PROGRAM LOADINGLOGIC
VAR
END_VAR


(*LOGIC TO DEFINE WHETHER THE MOBILE ATTACHMENT IS LOWERED PROPERLY IN THE GROUND*)
IF MOBILEHOIST.FLOORPOSITION_SWITCH1 AND MOBILEHOIST.FLOORPOSITION_SWITCH2 THEN
	
	MOBILEHOIST.LOWERED_PROPERLY 			:= TRUE;
	MOBILEHOIST.LOWERED_IMPROPERLY			:= FALSE;
	MOBILEHOIST.RAISED_PROPERLY				:= FALSE;
	
(*LOGIC TO DEFINE WHETHER THE MOBILE ATTACHMENT IS IMPROPERLY LOWERED*)	
ELSIF (MOBILEHOIST.FLOORPOSITION_SWITCH1 = FALSE AND MOBILEHOIST.FLOORPOSITION_SWITCH2) OR (MOBILEHOIST.FLOORPOSITION_SWITCH1 AND MOBILEHOIST.FLOORPOSITION_SWITCH2 = FALSE) THEN
	
	MOBILEHOIST.LOWERED_PROPERLY 			:= FALSE;
	MOBILEHOIST.LOWERED_IMPROPERLY			:= TRUE;
	MOBILEHOIST.RAISED_PROPERLY				:= FALSE;
	
ELSE
	
(*LOGIC TO DEFINE WHETHER THE MOBILE ATTACHMENT IS RAISED PROPERLY OF THE GROUND*)	
	IF (MOBILEHOIST.FLOORPOSITION_SWITCH1 = FALSE AND MOBILEHOIST.FLOORPOSITION_SWITCH2 = FALSE) THEN
		
	MOBILEHOIST.LOWERED_PROPERLY 			:= FALSE;
	MOBILEHOIST.LOWERED_IMPROPERLY			:= FALSE;
	MOBILEHOIST.RAISED_PROPERLY				:= TRUE;
		
	END_IF

END_IF

END_PROGRAM

(* stored: Version 1.1.0.1, ProductVersion 3.1.4024.11
   POU LOADINGLOGIC: Id {7a9bfe4f-e63c-462e-9063-134147b33325}, SpecialFunc None *)
